(* IEC 61131-3 sources: open62541_dart/test/plc/plc_programs/schneider_m240, 2 files *)

(* ---- GVL_Test.st ---- *)
// GVL_Test — OPC UA test fixture for Modicon M240 / M241 (EcoStruxure Machine
// Expert). SCALARS ONLY: the M240/M241 OPC UA server exposes flat symbols and
// cannot publish structured (DUT) types, so TestStruct is intentionally OMITTED
// here (matches supportsComplexTypes = false in ../../plc_config.dart).
//
// Mirrors test/plc/plc_fixture.dart. BrowseNames and IEC types below MUST NOT
// change; the tests resolve every node by BrowseName.
//
// Publishing is NOT done with pragmas on the M241 — you select these variables
// in the OPC UA Symbol Configuration in Machine Expert (see README.md).
// Paste this declaration into a Global Variable List named "GVL_Test".
VAR_GLOBAL
    // --- Scalars (read/write) ---------------------------------------------
    TestBool    : BOOL;                 // -> OPC UA Boolean
    TestInt     : INT;                  // 16-bit -> OPC UA Int16
    TestDint    : DINT;                 // 32-bit -> OPC UA Int32
    TestReal    : REAL;                 // float32 -> OPC UA Float
    TestLreal   : LREAL;                // float64 -> OPC UA Double
    TestString  : STRING;               // -> OPC UA String

    // --- Writable setpoint (REAL) -----------------------------------------
    Setpoint    : REAL;

    // --- Free-running liveness counter (DINT) -----------------------------
    // Incremented by PLC_PRG every cycle. Read-only from a client's view.
    Counter     : DINT;

    // --- Array[0..9] OF DINT (read/write) ---------------------------------
    TestArray   : ARRAY[0..9] OF DINT;
END_VAR

(* ---- PLC_PRG.st ---- *)
// PLC_PRG — cyclic program for the M240/M241 fixture.
// Assign this POU to a cyclic task (e.g. MAST) so Counter actually increments.
//
// Declaration part:
PROGRAM PLC_PRG
VAR
    bInit : BOOL := TRUE;
END_VAR

// Implementation part:
IF bInit THEN
    bInit := FALSE;
    GVL_Test.TestBool   := FALSE;
    GVL_Test.TestInt    := 0;
    GVL_Test.TestDint   := 0;
    GVL_Test.TestReal   := 0.0;
    GVL_Test.TestLreal  := 0.0;
    GVL_Test.TestString := '';
    GVL_Test.Setpoint   := 0.0;
    GVL_Test.Counter    := 0;
END_IF

// Liveness counter: increment every scan so clients can prove the program is
// running and measure read/subscription update timing. Wraps at the DINT limit.
GVL_Test.Counter := GVL_Test.Counter + 1;
